// TIA Portal V17 export
// export: Created 2024-09-02T12:50:28.8494477Z, ExportSetting WithDefaults, DisplayName Totally Integrated Automation Portal, DisplayVersion V17, DisplayName TIA Portal Openness, DisplayVersion V17, DisplayName TIA Portal Version Control Interface, DisplayVersion V17, DisplayName STEP 7 Professional, DisplayVersion V17, DisplayName STEP 7 Safety, DisplayVersion V17, DisplayName WinCC Professional, DisplayVersion V17
TYPE "TypeSKS_CAMERA"
// stored: IsFailsafeCompliant false
   STRUCT
      "A" { ExternalWritable := 'False'} : Struct
         Reset { ExternalWritable := 'False'} : Bool;
         RatePrg { ExternalWritable := 'False'} : Array[00..15] of Bool;
         StartPRG { ExternalWritable := 'False'} : Array[00..15] of Bool;
      END_STRUCT;
      H { ExternalWritable := 'False'} : Struct
         Reset { ExternalWritable := 'False'} : Bool;
         RatePrg { ExternalWritable := 'False'} : Array[00..15] of Bool;
         StartPRG { ExternalWritable := 'False'} : Array[00..15] of Bool;
      END_STRUCT;
   END_STRUCT;
END_TYPE
